(*

.. <legal notes>

legal notes
=================
| SPDX-FileCopyrightText: © 2026 Oleksandr Tiutyk <trofimich@gmail.com>
| SPDX-License-Identifier: LGPL-3.0-only
| For details check: LGPL-3.0-only_

.. _LGPL-3.0-only: https://www.gnu.org/licenses/lgpl-3.0.en.html

.. </legal notes>

*)

{attribute 'qualified_only'}
{attribute 'strict'}
{attribute 'to_string'}
TYPE INTERSECTION_STATE :
(
	ALL_OFF := 0,
	ALL_YELLOW,
	GROUP1_GREEN_GROUP2_RED,
	GROUP1_RED_GROUP2_GREEN
);
END_TYPE

(* stored: Version 1.1.0.1
   DUT INTERSECTION_STATE: Id {580c3efa-8e1c-4e07-a2f9-c98a0a6c9b11} *)
